// TwinCAT 3 PLC project Untitled1
// ProgramVersion: 3.1.4022.2
// libraries:
//   Tc2_Standard, * (Beckhoff Automation GmbH)
//   Tc2_System, * (Beckhoff Automation GmbH)
//   Tc3_EventLogger, * (Beckhoff Automation GmbH)
//   Tc3_Module, * (Beckhoff Automation GmbH)
// project tree:
//   / PlcTask.TcTTO (not stored)
//   POUs/ MAIN.TcPOU

// ---- POUs/MAIN.TcPOU
PROGRAM MAIN
VAR
	fbEventlogger : FB_TcEventLogger;
	fbAlarm: FB_TcAlarm;
	fbMessage: FB_TcMessage;
	
	bAlarm: BOOL;
	bMessage : BOOL;
	bIsInitalized: BOOL;
	bClearAlarm: BOOL;
	bConfirmAlarm: BOOL;
	
	fbCritical : FB_TcAlarm;
	fbSourceInfo : FB_TcSourceInfo;
	bCritical : BOOL;
END_VAR

IF NOT bIsInitalized THEN
	bIsInitalized := TRUE;
	
	fbMessage.CreateEx(TC_Events.MyEvents.Start, 0);
	fbAlarm.CreateEx(TC_Events.MyEvents.Stop, TRUE, 0);
	
	fbSourceInfo.Clear();
	fbSourceInfo.sName := 'Water pump 3'; 
	fbCritical.CreateEx(TC_EVENTS.MyEvents.Panic, TRUE, fbSourceInfo);
END_IF

IF bMessage THEN
	bMessage := FALSE;
	fbMessage.Send(0);
END_IF

IF bAlarm THEN
	bAlarm := FALSE;
	fbAlarm.Raise(0);
END_IF

IF bClearAlarm THEN
	bClearAlarm := FALSE;
	fbAlarm.Clear(0, TRUE);
END_IF

IF bCritical THEN
	bCritical := FALSE;
	fbCritical.Raise(0);
END_IF

END_PROGRAM
